Yaskawa INFORM job: R1_W49-52-A5(180,0)KM-OK.JBI

/JOB
//NAME R1_W49-52-A5(180,0)KM-OK
///FOLDERNAME KRIS-SCIANA
//POS
///NPOS 113,113,0,8,0,0
///TOOL 0
///POSTYPE PULSE
///PULSE
C00000=-197245,-85311,-91705,-27720,101707,32154
C00001=-222839,-80053,-84073,-30903,98416,38194
C00002=-222839,-80053,-84059,-30902,98409,38196
C00003=-224279,-80696,-84348,-30847,97757,37811
C00004=-222839,-80053,-84059,-30902,98409,38196
C00005=-222839,-80057,-83110,-30849,97904,38335
C00006=-222839,-80053,-84059,-30902,98409,38196
C00007=-211221,-87723,-86780,-30602,100653,42161
C00008=-211221,-87610,-85555,-30523,100052,42325
C00009=-211221,-87723,-86780,-30602,100653,42161
C00010=-241411,-126218,-117000,-4527,89497,34956
C00011=-241411,-126919,-112406,-4526,86317,35071
C00012=-241411,-125085,-111845,-4525,86913,35048
C00013=-241411,-126919,-112406,-4526,86317,35071
C00014=-241358,-132309,-117586,-4529,86739,35074
C00015=-193596,-91795,-99179,-7395,99760,50580
C00016=-196147,-90538,-97795,-7301,99329,49740
C00017=-196583,-89201,-97245,-7295,99637,49575
C00018=-196147,-90538,-97795,-7301,99329,49740
C00019=-196147,-89893,-100487,-7358,101301,49622
C00020=-202722,-67084,-90176,-7279,106068,47122
C00021=-202722,-69795,-83527,-7084,100623,47446
C00022=-202722,-69931,-82945,-7073,100198,47471
C00023=-202722,-69309,-85266,-7124,101933,47369
C00024=-188587,-66511,-91479,1998,102491,53492
C00025=-191000,-66345,-83583,2205,97780,52626
C00026=-191279,-65608,-83209,2235,97936,52537
C00027=-191000,-66345,-83583,2205,97780,52626
C00028=-191000,-65293,-86164,2221,99907,52664
C00029=-195913,-51178,-78584,2775,102636,51122
C00030=-195616,-54435,-73924,2696,98092,51118
C00031=-195616,-54573,-73481,2694,97747,51110
C00032=-195616,-54435,-73924,2696,98092,51118
C00033=-195616,-48301,-83837,2816,107333,51326
C00034=-189917,-32332,-65110,2161,103856,52837
C00035=-189917,-34069,-61967,2133,101029,52788
C00036=-189917,-34388,-61251,2130,100425,52777
C00037=-189917,-34742,-60383,2125,99710,52768
C00038=-189917,-34621,-60689,2127,99960,52772
C00039=-187742,-30911,-58233,1895,100303,53486
C00040=-187742,-31211,-57484,1893,99687,53479
C00041=-188522,-32565,-58388,1975,99564,53223
C00042=-188141,-31295,-59426,1929,100846,53363
C00043=-195712,-48687,-83670,2843,107033,51042
C00044=-225643,-91839,-90954,16656,91967,-41672
C00045=-225643,-89148,-77055,16645,85082,-42603
C00046=-222182,-87405,-73038,16450,82864,-41678
C00047=-220808,-86604,-71381,16368,82002,-41306
C00048=-220808,-86250,-70350,16384,81567,-41363
C00049=-220808,-86604,-71381,16368,82002,-41306
C00050=-219611,-86083,-71163,16272,81891,-40897
C00051=-221575,-86994,-71789,16422,82205,-41551
C00052=-217369,-94369,-76171,12335,77241,-39424
C00053=-219037,-94180,-73954,16325,79429,-41022
C00054=-219037,-93911,-73303,16337,79175,-41054
C00055=-219037,-94180,-73954,16325,79429,-41022
C00056=-217949,-93695,-73766,16233,79341,-40645
C00057=-219037,-94180,-73954,16325,79429,-41022
C00058=-220702,-97360,-80754,12690,79012,-40417
C00059=-224086,-90111,-72465,24610,81597,-25482
C00060=-224265,-87594,-68462,24684,80582,-25761
C00061=-225652,-76841,-67545,24645,88556,-18285
C00062=-226006,-87082,-67057,24810,80555,-26420
C00063=-224332,-87175,-68372,24678,80748,-25752
C00064=-225212,-79555,-67221,24641,86968,-18449
C00065=-224411,-82858,-66292,24664,84659,-18629
C00066=-225641,-71808,-60868,24566,91453,-31928
C00067=-224664,-71286,-59770,25306,95884,-30388
C00068=-224934,-80099,-63709,26004,90713,-27562
C00069=-226525,-84485,-64797,27782,88254,-27212
C00070=-224635,-80702,-62246,29506,93675,-25191
C00071=-225041,-80206,-60425,32862,88797,-44902
C00072=-225358,-79183,-62458,32869,90426,-44555
C00073=-228742,-68926,-72534,33620,101432,-42647
C00074=-229894,-66036,-88578,35838,111318,-39878
C00075=-229856,-65902,-88555,18555,100451,36555
C00076=-199408,-98171,-91827,-1508,74691,71158
C00077=-199283,-98682,-89760,-1556,73160,71223
C00078=-196273,-92715,-86732,-2354,74434,72254
C00079=-194004,-86541,-83203,-2946,75505,73018
C00080=-193898,-82965,-81939,-2963,76566,73026
C00081=-203929,-56131,-69140,6617,94917,70644
C00082=-195318,-66353,-72470,432,83590,72709
C00083=-191286,-71551,-73013,-3647,77046,73913
C00084=-191444,-70394,-72065,-3606,77052,73862
C00085=-181703,-53740,-63154,-14049,88170,75681
C00086=-188616,-43225,-56998,-11624,87635,73514
C00087=-196863,-64299,-73969,-2146,81160,71931
C00088=-208958,-93009,-95876,-5284,89959,67254
C00089=-206982,-92294,-92019,-6451,90245,67860
C00090=-200332,-81667,-86266,-7088,92702,69964
C00091=-207048,-92060,-94706,-6455,92002,67747
C00092=-227591,-113322,-106079,-4244,86735,61066
C00093=-227646,-113375,-102305,-4248,84388,61126
C00094=-218405,-105937,-98807,-5274,86600,64175
C00095=-218429,-106446,-105001,-5273,90133,64020
C00096=-213182,-106577,-100350,-5825,87576,65901
C00097=-222394,-112173,-102238,-4842,85261,62879
C00098=-222732,-112638,-104751,-4798,86545,62716
C00099=-234697,-116545,-106055,-3413,84733,58726
C00100=-235690,-116001,-103683,-3297,83514,58422
C00101=-231026,-112930,-101180,-12857,85384,59607
C00102=-222485,-100261,-98959,-13612,91784,61873
C00103=-206440,-114240,-97192,-28078,81592,53283
C00104=-219354,-57105,-77187,-20789,119054,64747
C00105=-225423,-62060,-74829,-20963,113825,63375
C00106=-218237,-99759,-89221,-22873,89467,47281
C00107=-217342,-103367,-87579,-26818,77697,50015
C00108=-221217,-81027,-78662,-25805,81871,47600
C00109=-208828,-90008,-86026,-27605,85759,51374
C00110=-229894,-53754,-99017,40266,121485,-35808
C00111=-140617,-50724,-97366,40349,121315,-35217
C00112=-139275,-147023,-123900,66598,-4025,-48175
BC00000=390625,1115520,1025624
BC00001=392319,1122406,1025764
BC00002=392319,1122406,1025764
BC00003=392319,1122406,1025764
BC00004=392319,1122406,1025764
BC00005=392319,1122406,1025764
BC00006=392319,1122406,1025764
BC00007=392319,1122406,1025764
BC00008=392319,1122406,1025764
BC00009=392319,1122406,1025764
BC00010=392319,1122406,1025764
BC00011=392319,1122406,1025764
BC00012=392320,1122407,1025761
BC00013=392319,1122406,1025764
BC00014=392319,1122406,1025764
BC00015=392319,1122406,1025764
BC00016=392319,1122406,1025764
BC00017=392319,1122406,1025764
BC00018=392319,1122406,1025764
BC00019=392319,1122406,1025764
BC00020=392319,1122406,1025764
BC00021=392319,1122406,1025764
BC00022=392319,1122406,1025764
BC00023=392319,1122406,1025764
BC00024=392319,1122406,1025764
BC00025=392319,1122406,1025762
BC00026=392319,1122406,1025762
BC00027=392319,1122406,1025762
BC00028=392319,1122406,1025762
BC00029=392319,1122406,1025762
BC00030=392319,1122406,1025762
BC00031=392319,1122406,1025762
BC00032=392319,1122406,1025762
BC00033=392319,1122406,1025762
BC00034=392329,1122535,1025762
BC00035=392329,1122535,1025762
BC00036=392329,1122535,1025762
BC00037=392329,1122535,1025762
BC00038=392329,1122535,1025762
BC00039=392329,1122535,1025762
BC00040=392329,1122535,1025762
BC00041=392329,1122535,1025762
BC00042=392328,1122534,1025760
BC00043=392329,1122535,1025762
BC00044=395849,1159283,1065533
BC00045=395849,1159283,1065533
BC00046=395849,1159283,1065533
BC00047=395849,1159283,1065533
BC00048=395849,1159283,1065533
BC00049=395849,1159283,1065533
BC00050=395849,1159283,1065533
BC00051=395849,1159283,1065533
BC00052=395849,1159283,1065533
BC00053=395849,1159283,1065533
BC00054=395849,1159283,1065533
BC00055=395849,1159283,1065533
BC00056=395849,1159283,1065533
BC00057=395849,1159283,1065533
BC00058=395849,1159283,1065533
BC00059=395849,1145308,1065533
BC00060=395849,1150672,1065533
BC00061=394411,1154217,1065532
BC00062=395849,1152817,1065533
BC00063=395849,1152817,1065533
BC00064=394411,1154217,1065532
BC00065=394411,1154217,1065532
BC00066=394410,1154219,1065533
BC00067=394410,1154219,1065533
BC00068=394410,1154219,1065533
BC00069=394410,1154219,1065533
BC00070=394410,1154219,1065533
BC00071=395849,1145456,1065533
BC00072=395849,1139585,1065533
BC00073=395849,1139585,1065533
BC00074=395849,1139585,1065533
BC00075=395846,1139570,1065499
BC00076=395846,1139570,1065499
BC00077=395846,1139570,1065499
BC00078=395846,1139570,1065499
BC00079=395846,1139570,1065499
BC00080=395846,1139570,1065499
BC00081=395846,1139570,1065499
BC00082=395846,1139570,1065499
BC00083=395846,1139570,1065499
BC00084=395846,1139570,1065499
BC00085=395846,1139570,1065499
BC00086=395846,1139570,1065499
BC00087=395846,1139570,1065499
BC00088=395846,1139570,1065499
BC00089=395846,1139570,1065499
BC00090=395846,1139570,1065499
BC00091=395846,1139570,1065499
BC00092=395846,1139570,1065499
BC00093=395846,1139570,1065499
BC00094=395846,1139570,1065499
BC00095=395846,1139570,1065499
BC00096=395846,1104918,1065499
BC00097=395846,1104918,1065499
BC00098=395846,1104918,1065499
BC00099=395846,1104918,1065499
BC00100=395846,1104918,1065499
BC00101=395846,1104918,1065499
BC00102=395846,1104918,1065499
BC00103=395846,1104918,1065499
BC00104=395846,1104918,1065499
BC00105=395846,1104918,1065499
BC00106=395846,1104918,1065496
BC00107=395846,1104918,1065499
BC00108=395846,1104918,1065499
BC00109=395846,1104918,1065499
BC00110=395849,1139585,1065533
BC00111=395849,1139585,1065533
BC00112=395849,1139585,1065533
///POSTYPE BASE
///RECTAN
///RCONF 0,0,0,0,0,0,0,0,0,0,0,0,0,0,0,0,0,0,0,0,0,0,0,0
P00006=0.222,-3.123,-1.508,0.0000,0.0000,0.0000
P00023=0.143,-0.036,0.682,0.0000,0.0000,0.0000
P00025=-2.003,0.006,0.728,0.0000,0.0000,0.0000
P00026=0.562,-0.002,-0.337,0.0000,0.0000,0.0000
P00027=-0.746,0.015,-9.096,0.0000,0.0000,0.0000
P00028=-2.237,-0.018,-7.702,0.0000,0.0000,0.0000
P00030=5.926,-4.294,-1.390,0.0000,0.0000,0.0000
P00050=4.296,-4.501,-0.826,0.0000,0.0000,0.0000
//INST
///DATE 2024/07/25 13:13
///ATTR SC,RW
///GROUP1 RB1,BS1
NOP
'r1_W49-52-A5(180,0)
'Path S1195
SFTOF
MOVJ C00000 BC00000 VJ=20.00
MOVJ C00001 BC00001 VJ=20.00
MOVL C00002 BC00002 V=83.3
REFP 3 C00003 BC00003
CALL JOB:SEARCH-R1
SET P025 P006
SFTON P025
MOVL C00004 BC00004 V=60.0
REFP 3 C00005 BC00005
CALL JOB:SEARCH-R1
SET P025 P006
SFTON P025
MOVL C00006 BC00006 V=60.0
SFTOF
MOVL C00007 BC00007 V=83.3
REFP 3 C00008 BC00008
CALL JOB:SEARCH-R1
SET P026 P006
SFTON P026
MOVL C00009 BC00009 V=83.3
MOVL C00010 BC00010 V=83.3
MOVL C00011 BC00011 V=83.3
REFP 3 C00012 BC00012
CALL JOB:SEARCH-R1
SET P026 P006
SFTON P026
MOVL C00013 BC00013 V=83.3
SFTOF
MOVL C00014 BC00014 V=83.3
MOVL C00015 BC00015 V=166.7
MOVL C00016 BC00016 V=83.3
REFP 3 C00017 BC00017
CALL JOB:SEARCH-R1
SET P027 P006
SFTON P027
MOVL C00018 BC00018 V=83.3
MOVL C00019 BC00019 V=83.3
MOVL C00020 BC00020 V=83.3
MOVL C00021 BC00021 V=83.3
REFP 3 C00022 BC00022
CALL JOB:SEARCH-R1
SET P027 P006
SFTON P027
MOVL C00023 BC00023 V=83.3
MOVL C00024 BC00024 V=166.7
SFTOF
MOVL C00025 BC00025 V=166.7
REFP 3 C00026 BC00026
CALL JOB:SEARCH-R1
SET P028 P006
SFTON P028
MOVL C00027 BC00027 V=83.3
MOVL C00028 BC00028 V=83.3
MOVL C00029 BC00029 V=83.3
MOVL C00030 BC00030 V=83.3
REFP 3 C00031 BC00031
CALL JOB:SEARCH-R1
SET P028 P006
SFTON P028
MOVL C00032 BC00032 V=83.3
MOVL C00033 BC00033 V=83.3
SFTOF
'BP 100624
MOVJ C00034 BC00034 VJ=25.00
MOVL C00035 BC00035 V=166.7
MOVL C00036 BC00036 V=60.0
REFP 3 C00037 BC00037
CALL JOB:SEARCH-R1
SET P050 P006
SFTON P050
MOVL C00038 BC00038 V=60.0
MOVL C00039 BC00039 V=166.7
MOVL C00040 BC00040 V=60.0
REFP 3 C00041 BC00041
CALL JOB:SEARCH-R1
SET P050 P006
SFTON P050
MOVL C00042 BC00042 V=166.7
SFTOF
'KONIEC BP 100624
MOVJ C00043 BC00043 VJ=25.00
MOVJ C00044 BC00044 VJ=25.00
MOVJ C00045 BC00045 VJ=10.00
MOVJ C00046 BC00046 VJ=10.00
MOVL C00047 BC00047 V=60.0
REFP 3 C00048 BC00048
CALL JOB:SEARCH-R1
SET P023 P006
SFTON P023
MOVL C00049 BC00049 V=60.0
REFP 3 C00050 BC00050
CALL JOB:SEARCH-R1
SET P023 P006
SFTON P023
MOVL C00051 BC00051 V=60.0
SFTOF
MOVL C00052 BC00052 V=100.0
MOVL C00053 BC00053 V=60.0
REFP 3 C00054 BC00054
CALL JOB:SEARCH-R1
SET P030 P006
SFTON P030
MOVL C00055 BC00055 V=60.0
REFP 3 C00056 BC00056
CALL JOB:SEARCH-R1
SET P030 P006
MOVL C00057 BC00057 V=60.0
MOVL C00058 BC00058 V=166.7
'Path W1196
SFTOF
SFTON P023
MOVJ C00059 BC00059 VJ=10.00
MOVJ C00060 BC00060 VJ=10.00
MOVL C00061 BC00061 V=100.0 PL=0
REFP 1 C00062 BC00062
REFP 2 C00063 BC00063
MACRO1 MJ#(0) ARGF9
ARCON
MOVL C00064 BC00064 V=10.0
MOVL C00065 BC00065 V=10.0
MOVL C00066 BC00066 V=9.2
SFTON P030
MOVL C00067 BC00067 V=9.2
MOVL C00068 BC00068 V=9.2
MOVL C00069 BC00069 V=9.2
MOVL C00070 BC00070 V=9.2
ARCOF
MOVL C00071 BC00071 V=166.7
MOVL C00072 BC00072 V=166.7
SFTOF
MOVJ C00073 BC00073 VJ=10.00
MOVJ C00074 BC00074 VJ=10.00
'SPAWANIE SPION PRZERYWANYCH
MOVJ C00075 BC00075 VJ=20.00
MACRO1 MJ#(0) ARGF6
MOVJ C00076 BC00076 VJ=20.00
SFTON P028
MOVJ C00077 BC00077 VJ=20.00
ARCON
MOVL C00078 BC00078 V=16.7
MOVL C00079 BC00079 V=16.7
ARCOF
MOVL C00080 BC00080 V=50.0
MOVL C00081 BC00081 V=50.0
ARCON
MOVL C00082 BC00082 V=11.7
MOVL C00083 BC00083 V=11.7
MACRO1 MJ#(0) ARGF6
ARCON
MACRO1 MJ#(0) ARGF6
MOVL C00084 BC00084 V=11.7
SFTON P050
MOVL C00085 BC00085 V=11.7
ARCON
WVON WEV#(50)
MACRO1 MJ#(0) ARGF12
MOVL C00086 BC00086 V=13.3
ARCOF
WVOF
MOVL C00087 BC00087 V=83.3
MACRO1 MJ#(0) ARGF6
MOVJ C00088 BC00088 VJ=20.00
SFTOF
SFTON P027
MOVJ C00089 BC00089 VJ=20.00
ARCON
MOVL C00090 BC00090 V=13.3
ARCOF
MOVJ C00091 BC00091 VJ=20.00
MOVJ C00092 BC00092 VJ=20.00
MOVJ C00093 BC00093 VJ=20.00
ARCON
MOVL C00094 BC00094 V=13.3
ARCOF
MOVJ C00095 BC00095 VJ=20.00
SFTOF
SFTON P026
MOVJ C00096 BC00096 VJ=20.00
ARCON
MOVL C00097 BC00097 V=13.3
ARCOF
MOVJ C00098 BC00098 VJ=20.00
MOVJ C00099 BC00099 VJ=20.00
MOVJ C00100 BC00100 VJ=20.00
ARCON
MOVL C00101 BC00101 V=16.7
ARCOF
MOVJ C00102 BC00102 VJ=20.00
SFTOF
MOVJ C00103 BC00103 VJ=20.00
MACRO1 MJ#(0) ARGF7
MOVJ C00104 BC00104 VJ=25.00
SFTON P025
MOVJ C00105 BC00105 VJ=20.00
ARCON
MOVL C00106 BC00106 V=8.3
MOVL C00107 BC00107 V=8.3
MOVL C00108 BC00108 V=8.3
ARCOF
MOVJ C00109 BC00109 VJ=20.00
SFTOF
MOVJ C00110 BC00110 VJ=10.00
MOVJ C00111 BC00111 VJ=50.00
MOVJ C00112 BC00112 VJ=100.00
SFTOF
END
